{attribute 'qualified_only'}
{attribute 'strict'}
TYPE E_BaseVisu :
(
	Idle := 0,
	Settings,
	Parameter,
	Manual,
	SemiAutomatic,
	Automatic,
	LogView
)INT;
END_TYPE

(* stored: Version 1.1.0.1, ProductVersion 3.1.4024.11
   EnumerationTextList E_BaseVisu: Id {f72244d6-971b-4c1b-8ca1-7c82c03cdf0f} *)
